// LS Electric XG5000 project: off delay
// PLC LSPLC
// module base 0 slot 0: 입력 모듈:XGI-D24A/B (DC 24V 입력, 32점 (전류소스 싱크공용/ 전류소스 입력))
// module base 0 slot 1: 출력 모듈:XGQ-TR4A/B (트랜지스터 출력, 32점 (0.1A용, 싱크출력/소스출력))

PROGRAM NewProgram (task: 스캔 프로그램)

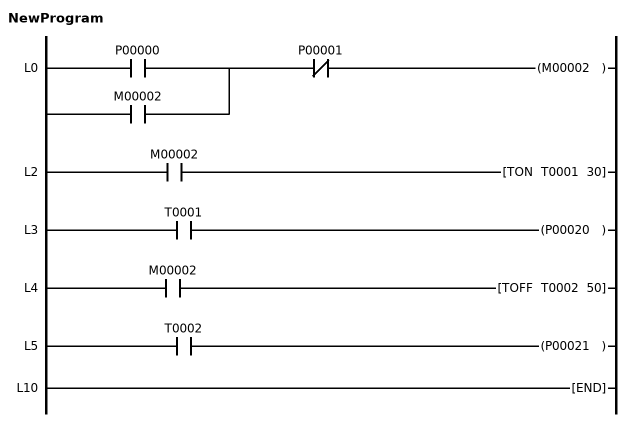
; L0
LOAD      P00000
OR        M00002
AND NOT   P00001
OUT       M00002
; L2
LOAD      M00002
TON       T0001 30
; L3
LOAD      T0001
OUT       P00020
; L4
LOAD      M00002
TOFF      T0002 50
; L5
LOAD      T0002
OUT       P00021
; L10
END